{attribute 'qualified_only'}
VAR_GLOBAL
//***********************************************************************************
//
// ETH Zürich / Robotic Fabrication Lab
// HIB C 13 / Stefano-Franscini-Platz 1
// CH-8093 Zürich
// 
// ***********************************************************************************
// 
// PROJECT     :  A061 Inline Mixer
// 
// FUNCTION    :  Global Varable to collect all research data
// 
// AUTHOR      :  Seyma Gürel / Philippe Fleischmann
// 
// EMAIL       :  scotto@arch.ethz.ch / fleischmann@arch.ehtz.ch
// 
// Copyright   :  ETH Zürich (CH) 2021
//
// ***********************************************************************************


// ***********************************************************************************
// Process inputs
// ***********************************************************************************

//
// Maximal speed for mixer [°/s]  
f_RED_Control_Speed : LREAL;					// [°/s]

//
// Accelerator Pump
b_RED_Acceleration_Pump_Calibration_On: BOOL;
n_RED_Acceleration_Pump_Calibration_Speed: INT;
n_RED_Acceleration_Pump_Calibration_Time: TIME;
f_RED_Acceleration_Pump_Mass: REAL;             // [g/min]
f_RED_Acceleration_Pump_Density: REAL;          // [g/ml]
n_RED_Acceleration_Pump_Flowrate: REAL;         // [ml/min]

//
// Concrete Pump
b_RED_Concrete_Pump_Forward_On: BOOL;
b_RED_Concrete_Pump_Backward_On: BOOL;
n_RED_Concrete_Pump_Speed: INT;					// [ 0..75rpm ]
		

// ***********************************************************************************
// Process outpus
// ***********************************************************************************

//
// Status mixer
b_RED_Status_On : BOOL;
f_RED_Status_Speed_Overide : LREAL;
f_RED_Status_Speed_Motor_1 : LREAL;
f_RED_Status_Speed_Motor_2 : LREAL;
f_RED_Status_Torque_Motor_1 : REAL;				// [Nm]
f_RED_Status_Torque_Motor_2 : REAL;				// [Nm]

// Weiting added 220817 
f_RED_Status_Temperature_Motor_1 : REAL; // [°C] 
f_RED_Status_Temperature_Motor_2 : REAL; // [°C] 

//
// Accelerator Pump
n_RED_Status_Acceleration_Pump_Flowrate: INT;          // [ml/min]
f_RED_Status_Acceleration_Pump_Max_Flowrate_ml_per_min: REAL;           // [ml/min]

END_VAR

(* stored: Version 1.1.0.1, ProductVersion 3.1.4024.2
   GVL GVL_ResearchData: Id {10f77899-a32f-44e6-ad7f-4be50514220e} *)
